// TIA Portal project "Erronka4" (V15.1)

(* hardware
DEVICE "S7-1200 station_1"  S7-1200 Station
   slot 0: "Rack_0"  S7-1200 Rack  Rack  V1.0
   slot 1: "PLC_1"  CPU 1214C AC/DC/Rly  6ES7 214-1BG40-0XB0  V4.0
   slot 3: "AQ 1x12BIT_1"  AQ1 signal board  6ES7 232-4HA30-0XB0  V1.0
*)

// ===== PLC "PLC_1"  CPU 1214C AC/DC/Rly =====

VAR_GLOBAL   // PLC tag table "Etapas"
   "Etapa0" AT %M16.0 : Bool;
   "Etapa1" AT %M16.1 : Bool;
   "Etapa2" AT %M16.2 : Bool;
   "Etapa3" AT %M16.3 : Bool;
   "Etapa4" AT %M16.4 : Bool;
   "Etapa5" AT %M16.5 : Bool;
   "Etapa6" AT %M16.6 : Bool;
   "Etapa7" AT %M16.7 : Bool;
   "Etapa8" AT %M17.0 : Bool;
   "Etapa9" AT %M17.1 : Bool;
   "Etapa20" AT %M20.0 : Bool;   // Inicio de STOP
   "Etapa21" AT %M20.1 : Bool;   // STOP
   "Etapa22" AT %M20.2 : Bool;   // STOP
   "MRMarca" AT %M90.0 : Bool;   // Marca del motor principal
   "Tag_2" AT %M302.0 : Bool;   // señal para ver si tenemos conexion
   "PE_Marca" AT %M300.0 : Bool;   // PE
   "RESET_PE_Marca" AT %M300.1 : Bool;   // PE
   "Tag_7" AT %MB302 : Byte;
   "DWetapas" AT %MD16 : DWord;   // Doble Word de las etapas
   "MDMotor" AT %MD90 : DWord;
   "Tag_10" AT %M50.0 : Bool;
   "Tag_12" AT %M50.1 : Bool;
   "TensionMotor" AT %MD70 : DWord;   // Tensión para mover MR
   "Tag_14" AT %MD74 : DWord;
   "CONTADORSALIDA" AT %MW100 : Int;
   "MARCAMOTORT" AT %M250.0 : Bool;
   "Tag_1" AT %MD250 : DWord;
END_VAR

VAR_GLOBAL   // PLC tag table "Entradas"
   "SDP1" AT %I0.1 : Bool;   // Sensor inductivo
   "SDP2" AT %I0.2 : Bool;   // Sensor (final de carrera)
   "SDP3" AT %I0.3 : Bool;   // Sensor con flanco de subida y bajada
   "SDP4" AT %I0.4 : Bool;   // Sensor magnetico en el cilindro CT
   "M" AT %I0.5 : Bool;   // Boton de marcha
   "PE" AT %I0.6 : Bool;   // Boton de para de emergencia
   "CR0" AT %I0.7 : Bool;   // Final de carrera CR0
   "CR1" AT %I1.0 : Bool;   // Final de carrera CR1
   "CT0" AT %I1.1 : Bool;   // Final de carrera CT0
   "CT1" AT %I1.2 : Bool;   // Final de carrera CT1
   "CC0" AT %I1.3 : Bool;   // Final de carrera CC0
   "CC1" AT %I1.4 : Bool;   // Final de carrera CC1
   "STOP" AT %I0.0 : Bool;   // Boton STOP
END_VAR

VAR_GLOBAL   // PLC tag table "Salidas"
   "MR" AT %Q2.4 : Bool;   // Motor principal
   "ACC" AT %Q0.1 : Bool;   // Aceleracion
   "DEC" AT %Q0.2 : Bool;   // Deceleracion
   "CR+" AT %Q0.3 : Bool;   // Salida del cilindro CR
   "CR-" AT %Q0.4 : Bool;   // Entrada del cilindro CR
   "CT+" AT %Q0.5 : Bool;   // Salida del cilindro CT
   "CT-" AT %Q0.6 : Bool;   // Entrada del cilindro CT
   "CC+" AT %Q0.7 : Bool;   // Salida del cilindro CC
   "CC-" AT %Q1.0 : Bool;   // Entrada del cilindro CC
   "MT" AT %Q1.1 : Bool;   // Motor Taladro
   "SEÑAL VARIADOR" AT %Q0.0 : Bool;   // Señal del Variador
   "Tag_16" AT %QW80 : Int;
END_VAR

// folder: System blocks/Program resources

DATA_BLOCK "Temporizador1"   // DB1
{ S7_Optimized_Access := 'TRUE' }
AUTHOR : Simatic
FAMILY : IEC
NAME : IEC_TMR
VERSION : 1.0
// stored: InstanceOfName IEC_TIMER
"IEC_TIMER"
BEGIN
END_DATA_BLOCK

DATA_BLOCK "Contador"   // DB3
{ S7_Optimized_Access := 'TRUE' }
AUTHOR : Simatic
FAMILY : IEC
NAME : CNTR
VERSION : 1.0
// stored: InstanceOfName IEC_COUNTER
"IEC_COUNTER"
BEGIN
END_DATA_BLOCK

// folder: (top level)

ORGANIZATION_BLOCK "Main"   // OB1, LAD, ProgramCycle
TITLE = "Main Program Sweep (Cycle)"
{ S7_Optimized_Access := 'TRUE' }
VERSION : 0.1
// En el main lo unico que hacemos es llamar a cada uno de los bloques de funciones que tenemos y estamos utilizando en este programa.
   VAR_INPUT
      Initial_Call : Bool;   // Initial call of this OB
      Remanence : Bool;   // =True, if remanent data are available
   END_VAR
BEGIN

REGION Network 1: MainGrafcet
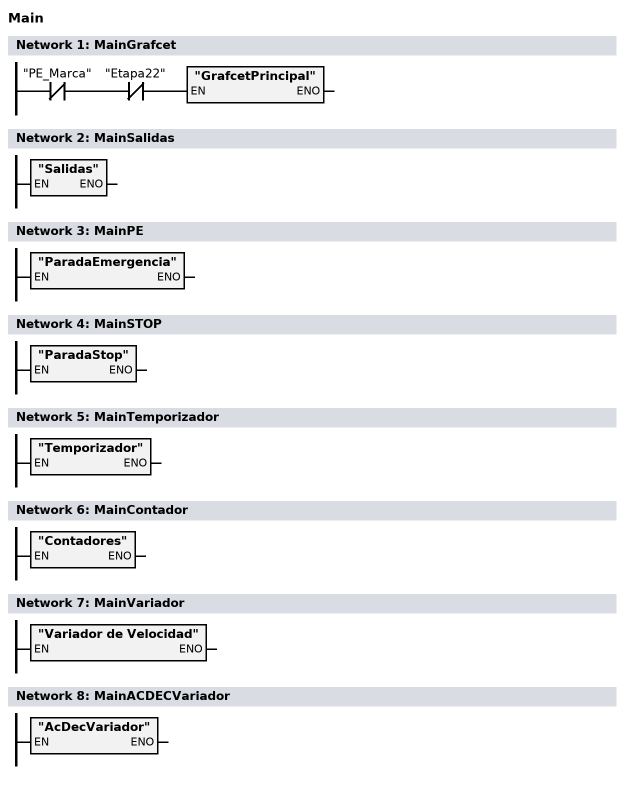
   RUNG wire#powerrail
      I_Contact( "PE_Marca" )
      I_Contact( "Etapa22" )
      "GrafcetPrincipal"()
   END_RUNG
   // the same network as SCL:
   IF NOT "PE_Marca" AND NOT "Etapa22" THEN "GrafcetPrincipal"(); END_IF;
END_REGION

REGION Network 2: MainSalidas
   RUNG wire#powerrail
      "Salidas"()
   END_RUNG
   // the same network as SCL:
   "Salidas"();
END_REGION

REGION Network 3: MainPE
   RUNG wire#powerrail
      "ParadaEmergencia"()
   END_RUNG
   // the same network as SCL:
   "ParadaEmergencia"();
END_REGION

REGION Network 4: MainSTOP
   RUNG wire#powerrail
      "ParadaStop"()
   END_RUNG
   // the same network as SCL:
   "ParadaStop"();
END_REGION

REGION Network 5: MainTemporizador
   RUNG wire#powerrail
      "Temporizador"()
   END_RUNG
   // the same network as SCL:
   "Temporizador"();
END_REGION

REGION Network 6: MainContador
   RUNG wire#powerrail
      "Contadores"()
   END_RUNG
   // the same network as SCL:
   "Contadores"();
END_REGION

REGION Network 7: MainVariador
   RUNG wire#powerrail
      "Variador de Velocidad"()
   END_RUNG
   // the same network as SCL:
   "Variador de Velocidad"();
END_REGION

REGION Network 8: MainACDECVariador
   RUNG wire#powerrail
      "AcDecVariador"()
   END_RUNG
   // the same network as SCL:
   "AcDecVariador"();
END_REGION
END_ORGANIZATION_BLOCK

ORGANIZATION_BLOCK "Startup"   // OB100, LAD, Startup
TITLE = "Complete Restart"
{ S7_Optimized_Access := 'TRUE' }
VERSION : 0.1
   VAR_INPUT
      LostRetentive : Bool;   // True if retentive data are lost
      LostRTC : Bool;   // True if date and time are lost
   END_VAR
BEGIN

REGION Network 1: Startup Etapa0
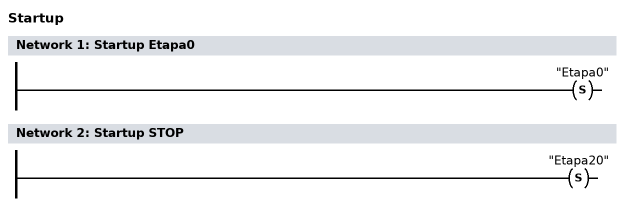
   RUNG wire#powerrail
      S_Coil( "Etapa0" )
   END_RUNG
   // the same network as SCL:
   "Etapa0" := TRUE;
END_REGION

REGION Network 2: Startup STOP
   RUNG wire#powerrail
      S_Coil( "Etapa20" )
   END_RUNG
   // the same network as SCL:
   "Etapa20" := TRUE;
END_REGION
END_ORGANIZATION_BLOCK

// folder: Funciones/FuncionBotonera

FUNCTION "ParadaStop" : Void   // FC2, LAD
TITLE = ParadaStop
{ S7_Optimized_Access := 'TRUE' }
VERSION : 0.1
// Esta todo lo relacionado con el stop
BEGIN

REGION Network 1: Etapa 20(stop)
   // La estapa 20 va a estar siempre activado por el startup o bien una vez ya se ha pausado el programa y pulsamos marcha para reanudarlo.
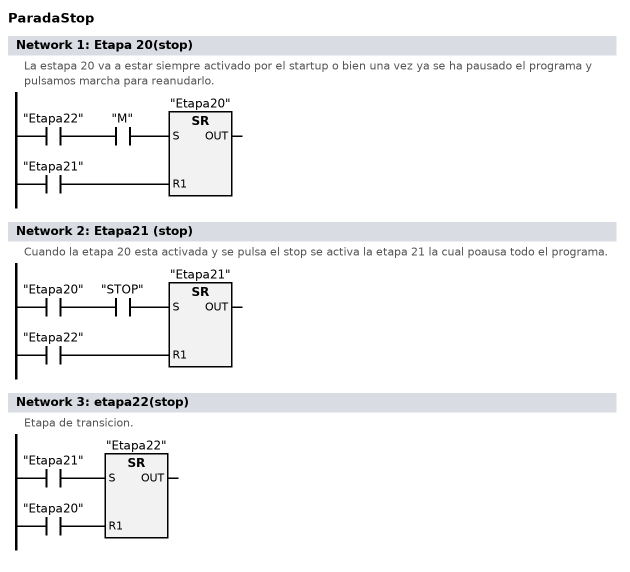
   RUNG wire#powerrail
      Contact( "Etapa22" )
      Contact( "M" )
      S_SR(operand := "Etapa20", r1 := wire#w1)
   END_RUNG
   RUNG wire#powerrail
      Contact( "Etapa21" )
   END_RUNG wire#w1
   // the same network as SCL:
   IF "Etapa22" AND "M" THEN
       "Etapa20" := TRUE;   // SR flip-flop
   END_IF;
   IF "Etapa21" THEN "Etapa20" := FALSE; END_IF;
END_REGION

REGION Network 2: Etapa21 (stop)
   // Cuando la etapa 20 esta activada y se pulsa el stop se activa la etapa 21 la cual poausa todo el programa.
   RUNG wire#powerrail
      Contact( "Etapa20" )
      Contact( "STOP" )
      S_SR(operand := "Etapa21", r1 := wire#w1)
   END_RUNG
   RUNG wire#powerrail
      Contact( "Etapa22" )
   END_RUNG wire#w1
   // the same network as SCL:
   IF "Etapa20" AND "STOP" THEN
       "Etapa21" := TRUE;   // SR flip-flop
   END_IF;
   IF "Etapa22" THEN "Etapa21" := FALSE; END_IF;
END_REGION

REGION Network 3: etapa22(stop)
   // Etapa de transicion.
   RUNG wire#powerrail
      Contact( "Etapa21" )
      S_SR(operand := "Etapa22", r1 := wire#w1)
   END_RUNG
   RUNG wire#powerrail
      Contact( "Etapa20" )
   END_RUNG wire#w1
   // the same network as SCL:
   IF "Etapa21" THEN
       "Etapa22" := TRUE;   // SR flip-flop
   END_IF;
   IF "Etapa20" THEN "Etapa22" := FALSE; END_IF;
END_REGION
END_FUNCTION

FUNCTION "ParadaEmergencia" : Void   // FC3, LAD
TITLE = ParadaEmergencia
{ S7_Optimized_Access := 'TRUE' }
VERSION : 0.1
// Esta todo lo relacionado con la parada de emergencia.
BEGIN

REGION Network 1: PE tag3
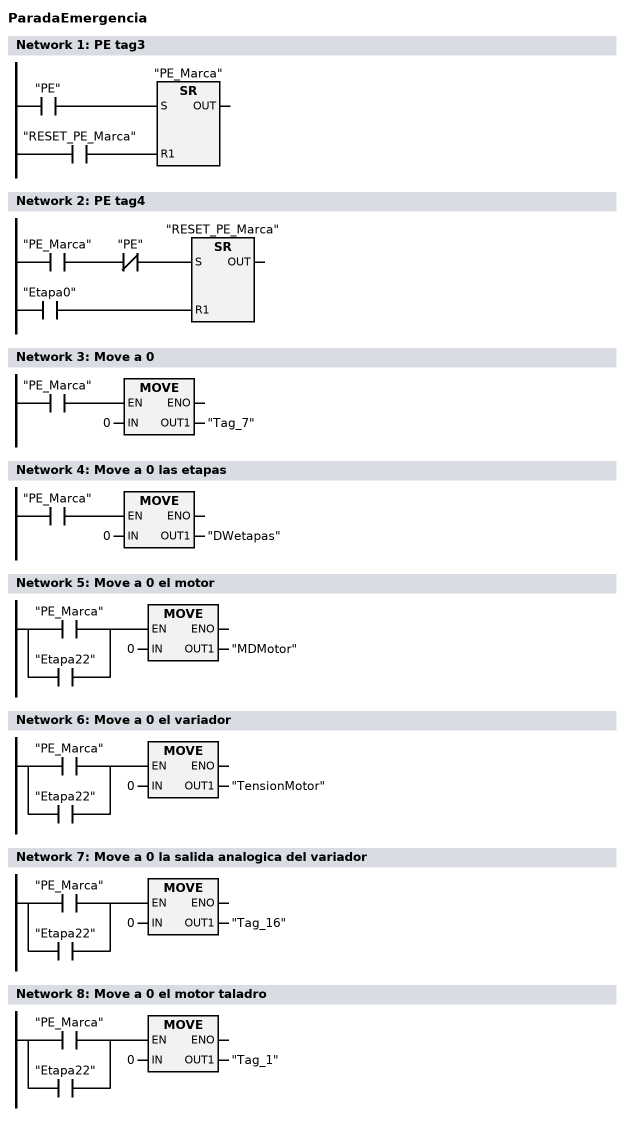
   RUNG wire#powerrail
      Contact( "PE" )
      S_SR(operand := "PE_Marca", r1 := wire#w1)
   END_RUNG
   RUNG wire#powerrail
      Contact( "RESET_PE_Marca" )
   END_RUNG wire#w1
   // the same network as SCL:
   IF "PE" THEN
       "PE_Marca" := TRUE;   // SR flip-flop
   END_IF;
   IF "RESET_PE_Marca" THEN "PE_Marca" := FALSE; END_IF;
END_REGION

REGION Network 2: PE tag4
   RUNG wire#powerrail
      Contact( "PE_Marca" )
      I_Contact( "PE" )
      S_SR(operand := "RESET_PE_Marca", r1 := wire#w1)
   END_RUNG
   RUNG wire#powerrail
      Contact( "Etapa0" )
   END_RUNG wire#w1
   // the same network as SCL:
   IF "PE_Marca" AND NOT "PE" THEN
       "RESET_PE_Marca" := TRUE;   // SR flip-flop
   END_IF;
   IF "Etapa0" THEN "RESET_PE_Marca" := FALSE; END_IF;
END_REGION

REGION Network 3: Move a 0
   RUNG wire#powerrail
      Contact( "PE_Marca" )
      Move(in := 0, out1 => "Tag_7")
   END_RUNG
   // the same network as SCL:
   IF "PE_Marca" THEN "Tag_7" := 0; END_IF;
END_REGION

REGION Network 4: Move a 0 las etapas
   RUNG wire#powerrail
      Contact( "PE_Marca" )
      Move(in := 0, out1 => "DWetapas")
   END_RUNG
   // the same network as SCL:
   IF "PE_Marca" THEN "DWetapas" := 0; END_IF;
END_REGION

REGION Network 5: Move a 0 el motor
   RUNG wire#powerrail
      Contact( "PE_Marca" )
      wire#w1
      Move(in := 0, out1 => "MDMotor")
   END_RUNG
   RUNG wire#powerrail
      Contact( "Etapa22" )
   END_RUNG wire#w1
   // the same network as SCL:
   IF "PE_Marca" OR "Etapa22" THEN "MDMotor" := 0; END_IF;
END_REGION

REGION Network 6: Move a 0 el variador
   RUNG wire#powerrail
      Contact( "PE_Marca" )
      wire#w1
      Move(in := 0, out1 => "TensionMotor")
   END_RUNG
   RUNG wire#powerrail
      Contact( "Etapa22" )
   END_RUNG wire#w1
   // the same network as SCL:
   IF "PE_Marca" OR "Etapa22" THEN "TensionMotor" := 0; END_IF;
END_REGION

REGION Network 7: Move a 0 la salida analogica del variador
   RUNG wire#powerrail
      Contact( "PE_Marca" )
      wire#w1
      Move(in := 0, out1 => "Tag_16")
   END_RUNG
   RUNG wire#powerrail
      Contact( "Etapa22" )
   END_RUNG wire#w1
   // the same network as SCL:
   IF "PE_Marca" OR "Etapa22" THEN "Tag_16" := 0; END_IF;
END_REGION

REGION Network 8: Move a 0 el motor taladro
   RUNG wire#powerrail
      Contact( "PE_Marca" )
      wire#w1
      Move(in := 0, out1 => "Tag_1")
   END_RUNG
   RUNG wire#powerrail
      Contact( "Etapa22" )
   END_RUNG wire#w1
   // the same network as SCL:
   IF "PE_Marca" OR "Etapa22" THEN "Tag_1" := 0; END_IF;
END_REGION
END_FUNCTION

// folder: Funciones/FuncionContador

FUNCTION "Contadores" : Void   // FC6, LAD
TITLE = Contadores
{ S7_Optimized_Access := 'TRUE' }
VERSION : 0.1
// Contador
BEGIN

REGION Network 1: Contador
   // Este es el contador el cual cuando llegue a 2 el programa se parara para poder contar las piezas. 
   // Se activa y cuenta con la etapa 8 guardandolo en una variable llamada contadorsalida y se resetea cuando llega a la etapa 0, que es o pulsando la para de emergencia o cuando ha hecho 2 veces el ciclo completo.
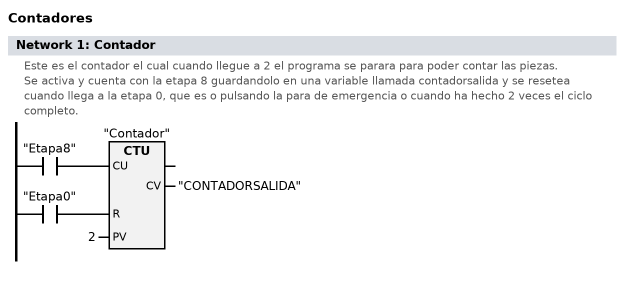
   "Contador".CTU(CU := "Etapa8", R := "Etapa0", PV := 2, CV => "CONTADORSALIDA");
END_REGION
END_FUNCTION

// folder: Funciones/FuncionGrafcet

FUNCTION "GrafcetPrincipal" : Void   // FC1, LAD
TITLE = GrafcetPrincipal
{ S7_Optimized_Access := 'TRUE' }
VERSION : 0.1
// Grafcet, programa base.
   VAR_TEMP   // added for the SCL form of the ladder/FBD networks
      _w1 : Bool;
   END_VAR
BEGIN

REGION Network 1: señal para ver si tenemos conexion
   // (Segmento creado para comprobar tras pulsar el boton de parada de emergencia que el FC1 
   // vuelve a estar funcional)
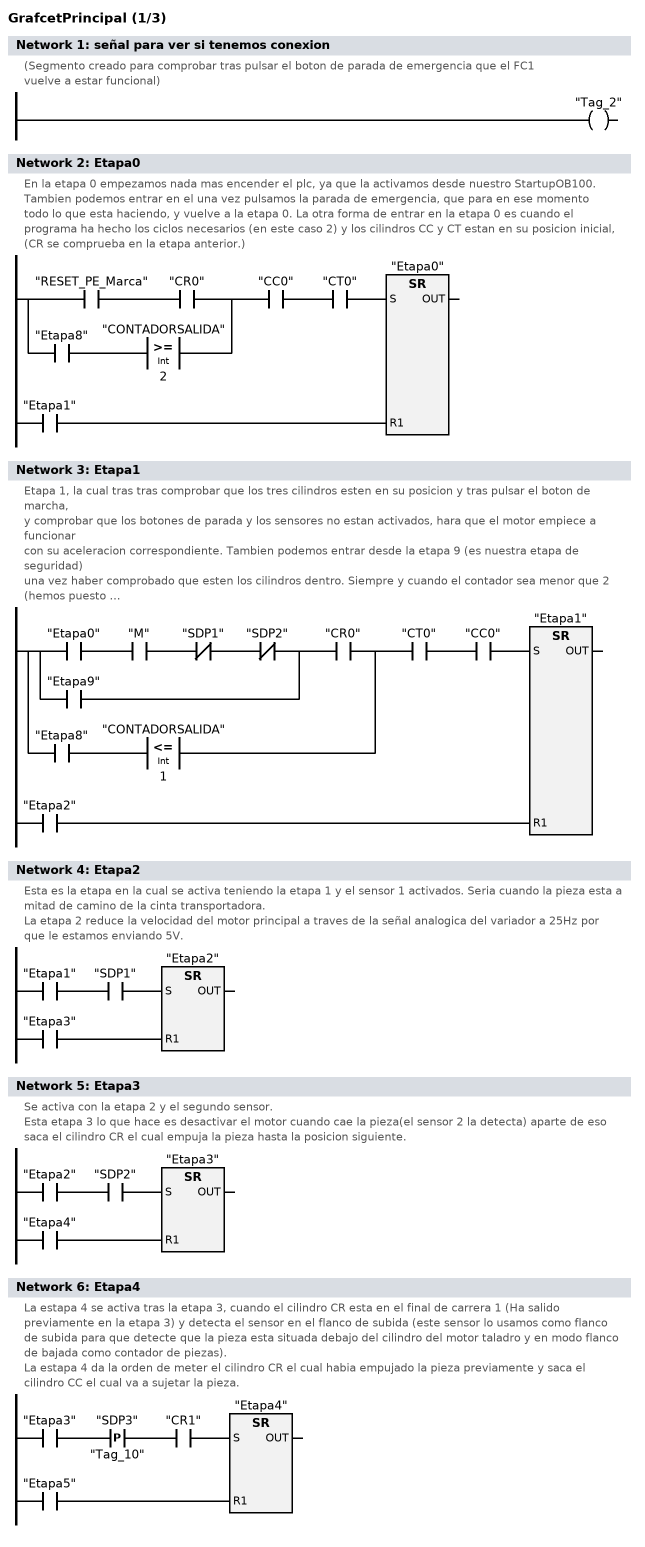
   RUNG wire#powerrail
      Coil( "Tag_2" )
   END_RUNG
   // the same network as SCL:
   "Tag_2" := TRUE;
END_REGION

REGION Network 2: Etapa0
   // En la etapa 0 empezamos nada mas encender el plc, ya que la activamos desde nuestro StartupOB100.
   // Tambien podemos entrar en el una vez pulsamos la parada de emergencia, que para en ese momento 
   // todo lo que esta haciendo, y vuelve a la etapa 0. La otra forma de entrar en la etapa 0 es cuando el 
   // programa ha hecho los ciclos necesarios (en este caso 2) y los cilindros CC y CT estan en su posicion inicial, (CR se comprueba en la etapa anterior.)
   RUNG wire#powerrail
      Contact( "RESET_PE_Marca" )
      Contact( "CR0" )
      wire#w1
      Contact( "CC0" )
      Contact( "CT0" )
      S_SR(operand := "Etapa0", r1 := wire#w2)
   END_RUNG
   RUNG wire#powerrail
      Contact( "Etapa8" )
      { S7_Templates := "SrcType := Int" } GE_Contact(in1 := "CONTADORSALIDA", in2 := 2)
   END_RUNG wire#w1
   RUNG wire#powerrail
      Contact( "Etapa1" )
   END_RUNG wire#w2
   // the same network as SCL:
   IF (("RESET_PE_Marca" AND "CR0") OR ("Etapa8" AND ("CONTADORSALIDA" >= 2))) AND "CC0" AND "CT0" THEN
       "Etapa0" := TRUE;   // SR flip-flop
   END_IF;
   IF "Etapa1" THEN "Etapa0" := FALSE; END_IF;
END_REGION

REGION Network 3: Etapa1
   // Etapa 1, la cual tras tras comprobar que los tres cilindros esten en su posicion y tras pulsar el boton de marcha, 
   // y comprobar que los botones de parada y los sensores no estan activados, hara que el motor empiece a funcionar
   // con su aceleracion correspondiente. Tambien podemos entrar desde la etapa 9 (es nuestra etapa de seguridad)
   // una vez haber comprobado que esten los cilindros dentro. Siempre y cuando el contador sea menor que 2 (hemos puesto 2 
   // en vez de 10 ya que era mas visual) tambien activaremos la etapa1.
   // 
   // La etapa 1 enciende el motor principal  a traves de la señal analogica del variador a 50Hz por que le estamos enviando 10V.
   RUNG wire#powerrail
      Contact( "Etapa0" )
      Contact( "M" )
      I_Contact( "SDP1" )
      I_Contact( "SDP2" )
      wire#w1
      Contact( "CR0" )
      wire#w2
      Contact( "CT0" )
      Contact( "CC0" )
      S_SR(operand := "Etapa1", r1 := wire#w3)
   END_RUNG
   RUNG wire#powerrail
      Contact( "Etapa9" )
   END_RUNG wire#w1
   RUNG wire#powerrail
      Contact( "Etapa8" )
      { S7_Templates := "SrcType := Int" } LE_Contact(in1 := "CONTADORSALIDA", in2 := 1)
   END_RUNG wire#w2
   RUNG wire#powerrail
      Contact( "Etapa2" )
   END_RUNG wire#w3
   // the same network as SCL:
   IF (((("Etapa0" AND "M" AND NOT "SDP1" AND NOT "SDP2") OR "Etapa9") AND "CR0") OR ("Etapa8" AND ("CONTADORSALIDA" <= 1))) AND "CT0" AND "CC0" THEN
       "Etapa1" := TRUE;   // SR flip-flop
   END_IF;
   IF "Etapa2" THEN "Etapa1" := FALSE; END_IF;
END_REGION

REGION Network 4: Etapa2
   // Esta es la etapa en la cual se activa teniendo la etapa 1 y el sensor 1 activados. Seria cuando la pieza esta a mitad de camino de la cinta transportadora.
   // 
   // La etapa 2 reduce la velocidad del motor principal a traves de la señal analogica del variador a 25Hz por que le estamos enviando 5V.
   RUNG wire#powerrail
      Contact( "Etapa1" )
      Contact( "SDP1" )
      S_SR(operand := "Etapa2", r1 := wire#w1)
   END_RUNG
   RUNG wire#powerrail
      Contact( "Etapa3" )
   END_RUNG wire#w1
   // the same network as SCL:
   IF "Etapa1" AND "SDP1" THEN
       "Etapa2" := TRUE;   // SR flip-flop
   END_IF;
   IF "Etapa3" THEN "Etapa2" := FALSE; END_IF;
END_REGION

REGION Network 5: Etapa3
   // Se activa con la etapa 2 y el segundo sensor.
   // 
   // Esta etapa 3 lo que hace es desactivar el motor cuando cae la pieza(el sensor 2 la detecta) aparte de eso saca el cilindro CR el cual empuja la pieza hasta la posicion siguiente.
   RUNG wire#powerrail
      Contact( "Etapa2" )
      Contact( "SDP2" )
      S_SR(operand := "Etapa3", r1 := wire#w1)
   END_RUNG
   RUNG wire#powerrail
      Contact( "Etapa4" )
   END_RUNG wire#w1
   // the same network as SCL:
   IF "Etapa2" AND "SDP2" THEN
       "Etapa3" := TRUE;   // SR flip-flop
   END_IF;
   IF "Etapa4" THEN "Etapa3" := FALSE; END_IF;
END_REGION

REGION Network 6: Etapa4
   // La estapa 4 se activa tras la etapa 3, cuando el cilindro CR esta en el final de carrera 1 (Ha salido previamente en la etapa 3) y detecta el sensor en el flanco de subida (este sensor lo usamos como flanco de subida para que detecte que la pieza esta situada debajo del cilindro del motor taladro y en modo flanco de bajada como contador de piezas).
   // 
   // La estapa 4 da la orden de meter el cilindro CR el cual habia empujado la pieza previamente y saca el cilindro CC el cual va a sujetar la pieza.
   RUNG wire#powerrail
      Contact( "Etapa3" )
      P_Contact(operand := "SDP3", bit := "Tag_10")
      Contact( "CR1" )
      S_SR(operand := "Etapa4", r1 := wire#w1)
   END_RUNG
   RUNG wire#powerrail
      Contact( "Etapa5" )
   END_RUNG wire#w1
   // the same network as SCL:
   #_w1 := "Etapa3" AND "SDP3" AND NOT "Tag_10";   // rising edge of "SDP3"
   "Tag_10" := "SDP3";
   IF #_w1 AND "CR1" THEN
       "Etapa4" := TRUE;   // SR flip-flop
   END_IF;
   IF "Etapa5" THEN "Etapa4" := FALSE; END_IF;
END_REGION

REGION Network 7: Etapa5
   // Se activa con la etapa4, cuando el cilindro CR ha vuelto y el cilindro CC que es el que sujeta la pieza.
   // 
   // La funcion de la etapa 5 es sacar el cilindro CT que es el cual va a taladrar la pieza.
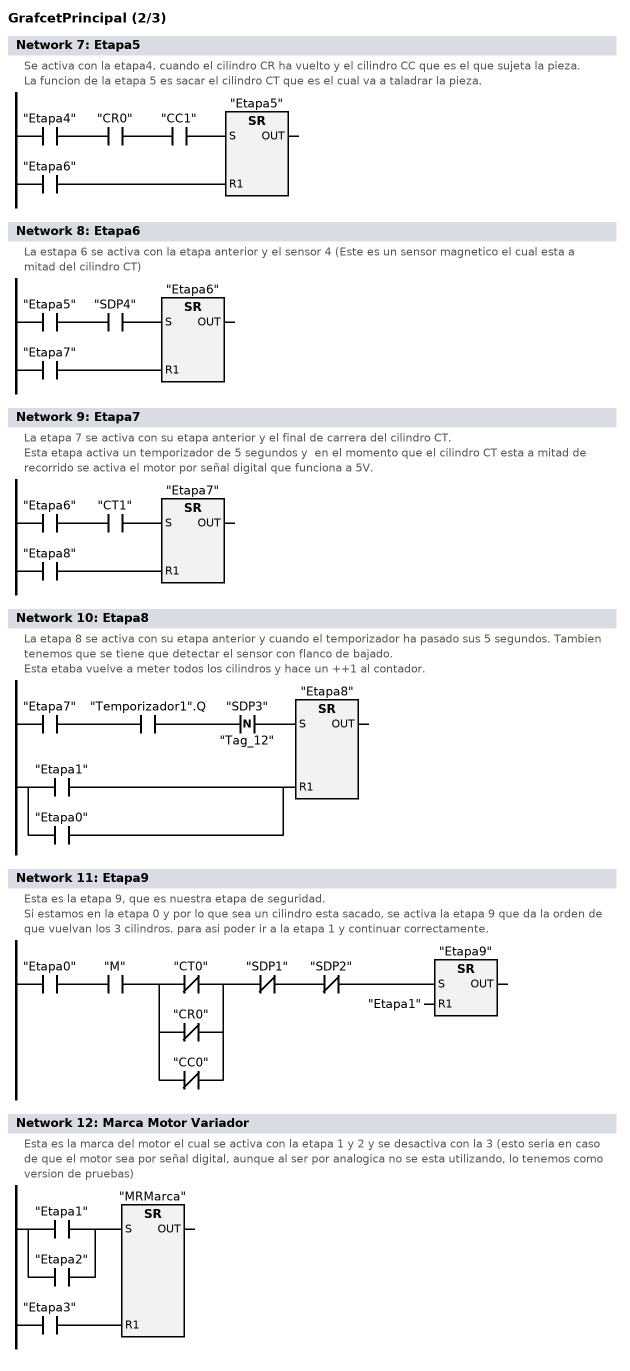
   RUNG wire#powerrail
      Contact( "Etapa4" )
      Contact( "CR0" )
      Contact( "CC1" )
      S_SR(operand := "Etapa5", r1 := wire#w1)
   END_RUNG
   RUNG wire#powerrail
      Contact( "Etapa6" )
   END_RUNG wire#w1
   // the same network as SCL:
   IF "Etapa4" AND "CR0" AND "CC1" THEN
       "Etapa5" := TRUE;   // SR flip-flop
   END_IF;
   IF "Etapa6" THEN "Etapa5" := FALSE; END_IF;
END_REGION

REGION Network 8: Etapa6
   // La estapa 6 se activa con la etapa anterior y el sensor 4 (Este es un sensor magnetico el cual esta a mitad del cilindro CT)
   RUNG wire#powerrail
      Contact( "Etapa5" )
      Contact( "SDP4" )
      S_SR(operand := "Etapa6", r1 := wire#w1)
   END_RUNG
   RUNG wire#powerrail
      Contact( "Etapa7" )
   END_RUNG wire#w1
   // the same network as SCL:
   IF "Etapa5" AND "SDP4" THEN
       "Etapa6" := TRUE;   // SR flip-flop
   END_IF;
   IF "Etapa7" THEN "Etapa6" := FALSE; END_IF;
END_REGION

REGION Network 9: Etapa7
   // La etapa 7 se activa con su etapa anterior y el final de carrera del cilindro CT.
   // 
   // Esta etapa activa un temporizador de 5 segundos y  en el momento que el cilindro CT esta a mitad de recorrido se activa el motor por señal digital que funciona a 5V.
   RUNG wire#powerrail
      Contact( "Etapa6" )
      Contact( "CT1" )
      S_SR(operand := "Etapa7", r1 := wire#w1)
   END_RUNG
   RUNG wire#powerrail
      Contact( "Etapa8" )
   END_RUNG wire#w1
   // the same network as SCL:
   IF "Etapa6" AND "CT1" THEN
       "Etapa7" := TRUE;   // SR flip-flop
   END_IF;
   IF "Etapa8" THEN "Etapa7" := FALSE; END_IF;
END_REGION

REGION Network 10: Etapa8
   // La etapa 8 se activa con su etapa anterior y cuando el temporizador ha pasado sus 5 segundos. Tambien tenemos que se tiene que detectar el sensor con flanco de bajado.
   // 
   // Esta etaba vuelve a meter todos los cilindros y hace un ++1 al contador.
   RUNG wire#powerrail
      Contact( "Etapa7" )
      Contact( "Temporizador1".Q )
      N_Contact(operand := "SDP3", bit := "Tag_12")
      S_SR(operand := "Etapa8", r1 := wire#w1)
   END_RUNG
   RUNG wire#powerrail
      Contact( "Etapa1" )
   END_RUNG wire#w1
   RUNG wire#powerrail
      Contact( "Etapa0" )
   END_RUNG wire#w1
   // the same network as SCL:
   #_w1 := "Etapa7" AND "Temporizador1".Q AND NOT "SDP3" AND "Tag_12";   // falling edge of "SDP3"
   "Tag_12" := "SDP3";
   IF #_w1 THEN
       "Etapa8" := TRUE;   // SR flip-flop
   END_IF;
   IF "Etapa1" OR "Etapa0" THEN "Etapa8" := FALSE; END_IF;
END_REGION

REGION Network 11: Etapa9
   // Esta es la etapa 9, que es nuestra etapa de seguridad.
   // Si estamos en la etapa 0 y por lo que sea un cilindro esta sacado, se activa la etapa 9 que da la orden de que vuelvan los 3 cilindros. para asi poder ir a la etapa 1 y continuar correctamente.
   RUNG wire#powerrail
      Contact( "Etapa0" )
      Contact( "M" )
      wire#w1
      I_Contact( "CT0" )
      wire#w2
      I_Contact( "SDP1" )
      I_Contact( "SDP2" )
      S_SR(operand := "Etapa9", r1 := "Etapa1")
   END_RUNG
   RUNG wire#w1
      I_Contact( "CR0" )
   END_RUNG wire#w2
   RUNG wire#w1
      I_Contact( "CC0" )
   END_RUNG wire#w2
   // the same network as SCL:
   IF "Etapa0" AND "M" AND (NOT "CT0" OR NOT "CR0" OR NOT "CC0") AND NOT "SDP1" AND NOT "SDP2" THEN
       "Etapa9" := TRUE;   // SR flip-flop
   END_IF;
   IF "Etapa1" THEN "Etapa9" := FALSE; END_IF;
END_REGION

REGION Network 12: Marca Motor Variador
   // Esta es la marca del motor el cual se activa con la etapa 1 y 2 y se desactiva con la 3 (esto seria en caso de que el motor sea por señal digital, aunque al ser por analogica no se esta utilizando, lo tenemos como version de pruebas)
   RUNG wire#powerrail
      Contact( "Etapa1" )
      wire#w1
      S_SR(operand := "MRMarca", r1 := wire#w2)
   END_RUNG
   RUNG wire#powerrail
      Contact( "Etapa2" )
   END_RUNG wire#w1
   RUNG wire#powerrail
      Contact( "Etapa3" )
   END_RUNG wire#w2
   // the same network as SCL:
   IF "Etapa1" OR "Etapa2" THEN
       "MRMarca" := TRUE;   // SR flip-flop
   END_IF;
   IF "Etapa3" THEN "MRMarca" := FALSE; END_IF;
END_REGION

REGION Network 13
   // esta es la marca del motor taladro la cual se activa con la etapa 6 y 7.
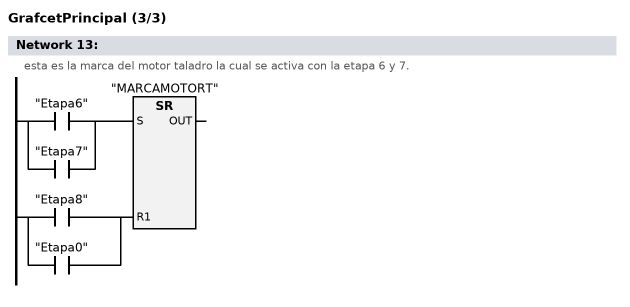
   RUNG wire#powerrail
      Contact( "Etapa6" )
      wire#w1
      S_SR(operand := "MARCAMOTORT", r1 := wire#w2)
   END_RUNG
   RUNG wire#powerrail
      Contact( "Etapa7" )
   END_RUNG wire#w1
   RUNG wire#powerrail
      Contact( "Etapa8" )
   END_RUNG wire#w2
   RUNG wire#powerrail
      Contact( "Etapa0" )
   END_RUNG wire#w2
   // the same network as SCL:
   IF "Etapa6" OR "Etapa7" THEN
       "MARCAMOTORT" := TRUE;   // SR flip-flop
   END_IF;
   IF "Etapa8" OR "Etapa0" THEN "MARCAMOTORT" := FALSE; END_IF;
END_REGION
END_FUNCTION

// folder: Funciones/FuncionSalidas

FUNCTION "Salidas" : Void   // FC4, LAD
TITLE = Salidas
{ S7_Optimized_Access := 'TRUE' }
VERSION : 0.1
// Salidas
BEGIN

REGION Network 1: SalidaMotor
   // Marca que activa el motor(no se usa en el programa ya que va con el variador, son pruebas para comprobar que todo funcione a la perfeccion.)
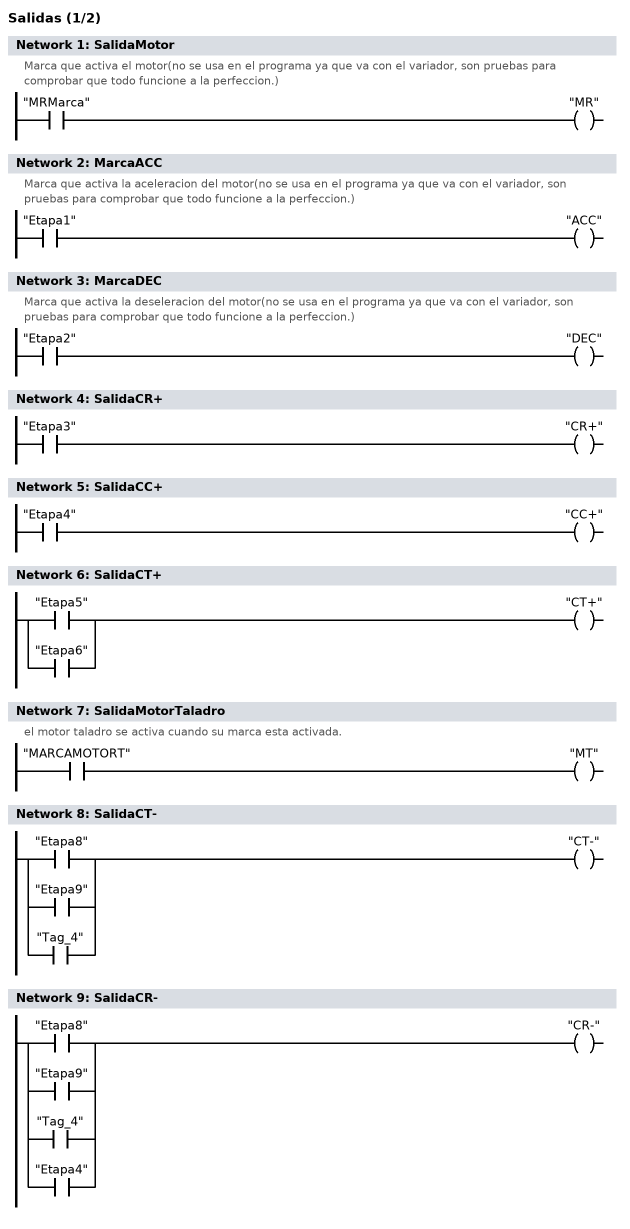
   RUNG wire#powerrail
      Contact( "MRMarca" )
      Coil( "MR" )
   END_RUNG
   // the same network as SCL:
   "MR" := "MRMarca";
END_REGION

REGION Network 2: MarcaACC
   // Marca que activa la aceleracion del motor(no se usa en el programa ya que va con el variador, son pruebas para comprobar que todo funcione a la perfeccion.)
   RUNG wire#powerrail
      Contact( "Etapa1" )
      Coil( "ACC" )
   END_RUNG
   // the same network as SCL:
   "ACC" := "Etapa1";
END_REGION

REGION Network 3: MarcaDEC
   // Marca que activa la deseleracion del motor(no se usa en el programa ya que va con el variador, son pruebas para comprobar que todo funcione a la perfeccion.)
   RUNG wire#powerrail
      Contact( "Etapa2" )
      Coil( "DEC" )
   END_RUNG
   // the same network as SCL:
   "DEC" := "Etapa2";
END_REGION

REGION Network 4: SalidaCR+
   RUNG wire#powerrail
      Contact( "Etapa3" )
      Coil( "CR+" )
   END_RUNG
   // the same network as SCL:
   "CR+" := "Etapa3";
END_REGION

REGION Network 5: SalidaCC+
   RUNG wire#powerrail
      Contact( "Etapa4" )
      Coil( "CC+" )
   END_RUNG
   // the same network as SCL:
   "CC+" := "Etapa4";
END_REGION

REGION Network 6: SalidaCT+
   RUNG wire#powerrail
      Contact( "Etapa5" )
      wire#w1
      Coil( "CT+" )
   END_RUNG
   RUNG wire#powerrail
      Contact( "Etapa6" )
   END_RUNG wire#w1
   // the same network as SCL:
   "CT+" := "Etapa5" OR "Etapa6";
END_REGION

REGION Network 7: SalidaMotorTaladro
   // el motor taladro se activa cuando su marca esta activada.
   RUNG wire#powerrail
      Contact( "MARCAMOTORT" )
      Coil( "MT" )
   END_RUNG
   // the same network as SCL:
   "MT" := "MARCAMOTORT";
END_REGION

REGION Network 8: SalidaCT-
   RUNG wire#powerrail
      Contact( "Etapa8" )
      wire#w1
      Coil( "CT-" )
   END_RUNG
   RUNG wire#powerrail
      Contact( "Etapa9" )
   END_RUNG wire#w1
   RUNG wire#powerrail
      Contact( "Tag_4" )
   END_RUNG wire#w1
   // the same network as SCL:
   "CT-" := "Etapa8" OR "Etapa9" OR "Tag_4";
END_REGION

REGION Network 9: SalidaCR-
   RUNG wire#powerrail
      Contact( "Etapa8" )
      wire#w1
      Coil( "CR-" )
   END_RUNG
   RUNG wire#powerrail
      Contact( "Etapa9" )
   END_RUNG wire#w1
   RUNG wire#powerrail
      Contact( "Tag_4" )
   END_RUNG wire#w1
   RUNG wire#powerrail
      Contact( "Etapa4" )
   END_RUNG wire#w1
   // the same network as SCL:
   "CR-" := "Etapa8" OR "Etapa9" OR "Tag_4" OR "Etapa4";
END_REGION

REGION Network 10: SalidaCC-
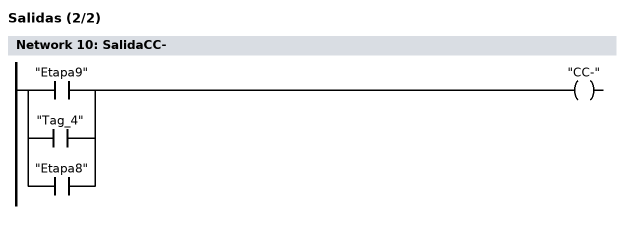
   RUNG wire#powerrail
      Contact( "Etapa9" )
      wire#w1
      Coil( "CC-" )
   END_RUNG
   RUNG wire#powerrail
      Contact( "Tag_4" )
   END_RUNG wire#w1
   RUNG wire#powerrail
      Contact( "Etapa8" )
   END_RUNG wire#w1
   // the same network as SCL:
   "CC-" := "Etapa9" OR "Tag_4" OR "Etapa8";
END_REGION
END_FUNCTION

// folder: Funciones/FuncionTemporizador

FUNCTION "Temporizador" : Void   // FC5, LAD
TITLE = Temporizador
{ S7_Optimized_Access := 'TRUE' }
VERSION : 0.1
// Temporizador
BEGIN

REGION Network 1: Temporizador
   // Este es el temporizador que cuenta los 5 segundos que esta taladrando el motor.
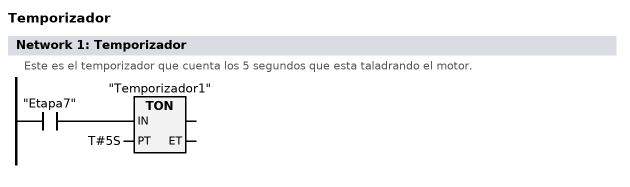
   "Temporizador1".TON(IN := "Etapa7", PT := T#5S);
END_REGION
END_FUNCTION

// folder: Funciones/FuncionVariador

FUNCTION "Variador de Velocidad" : Void   // FC7, LAD
TITLE = Variador
{ S7_Optimized_Access := 'TRUE' }
VERSION : 0.1
// Variador
BEGIN

REGION Network 1: NORM_X / SCALE_X (Variador)
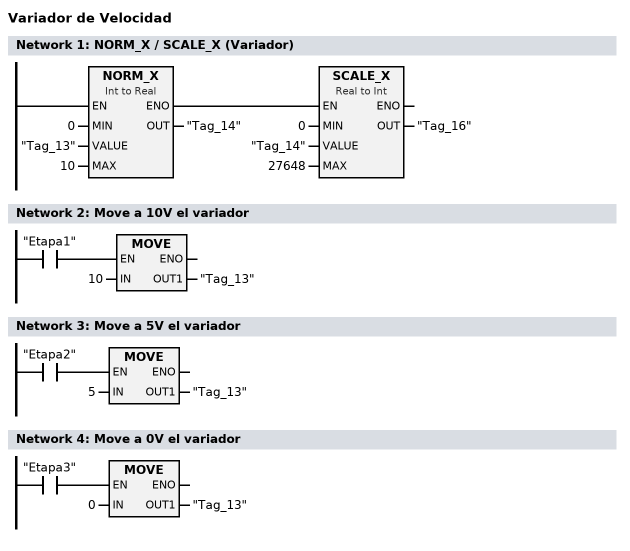
   RUNG wire#powerrail
      { S7_Templates := "[SrcType := Int, DestType := Real]" } Normalize(min := 0, value := "Tag_13", max := 10, out => "Tag_14")
      { S7_Templates := "[SrcType := Real, DestType := Int]" } Scale(min := 0, value := "Tag_14", max := 27648, out => "Tag_16")
   END_RUNG
   // the same network as SCL:
   "Tag_14" := NORM_X(MIN := 0, VALUE := "Tag_13", MAX := 10);
   "Tag_16" := SCALE_X(MIN := 0, VALUE := "Tag_14", MAX := 27648);
END_REGION

REGION Network 2: Move a 10V el variador
   RUNG wire#powerrail
      Contact( "Etapa1" )
      Move(in := 10, out1 => "Tag_13")
   END_RUNG
   // the same network as SCL:
   IF "Etapa1" THEN "Tag_13" := 10; END_IF;
END_REGION

REGION Network 3: Move a 5V el variador
   RUNG wire#powerrail
      Contact( "Etapa2" )
      Move(in := 5, out1 => "Tag_13")
   END_RUNG
   // the same network as SCL:
   IF "Etapa2" THEN "Tag_13" := 5; END_IF;
END_REGION

REGION Network 4: Move a 0V el variador
   RUNG wire#powerrail
      Contact( "Etapa3" )
      Move(in := 0, out1 => "Tag_13")
   END_RUNG
   // the same network as SCL:
   IF "Etapa3" THEN "Tag_13" := 0; END_IF;
END_REGION
END_FUNCTION

FUNCTION "AcDecVariador" : Void   // FC8, LAD
TITLE = SeñalVariador
{ S7_Optimized_Access := 'TRUE' }
VERSION : 0.1
// SeñalVariador
BEGIN

REGION Network 1: SeñalVariador
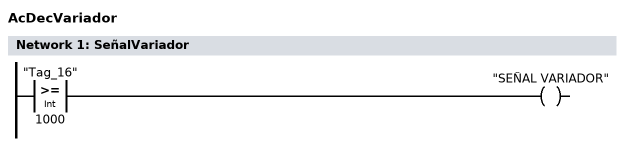
   RUNG wire#powerrail
      { S7_Templates := "SrcType := Int" } GE_Contact(in1 := "Tag_16", in2 := 1000)
      Coil( "SEÑAL VARIADOR" )
   END_RUNG
   // the same network as SCL:
   "SEÑAL VARIADOR" := "Tag_16" >= 1000;
END_REGION
END_FUNCTION